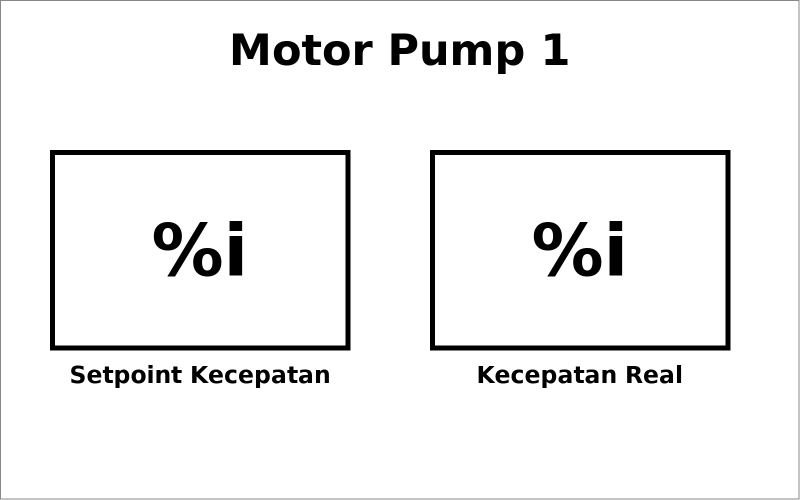
VISUALIZATION Screen_2_Sub_3  // 800x500
    Label (0,0 800x100), "Motor Pump 1"
    Rectangle (50,150 300x200), "%i", text variable: GVL.HMI_Motor_Pump_1_Input
        OnMouseClick: write GVL.HMI_Motor_Pump_1_Input via VisuDialogs.Numpad
    Label (50,350 300x50), "Setpoint Kecepatan"
    Label (430,350 300x50), "Kecepatan Real"
    Rectangle (430,150 300x200), "%i", text variable: GVL.HMI_Motor_Pump_1_Real
END_VISUALIZATION

(* stored: Version 1.1.0.1, ProductVersion 3.1.4024.12
   Visu Screen_2_Sub_3: Id {79021551-012e-4111-94d3-d65a07dec9a8} *)
